	//Device Information Parameter
	_strDeviceCode		: STRING(51);		// Hardware Version Name from Device read acyclic	
	//Values read with acyclic FB
	_rTemperature		: REAL;				//24 P0-09 Heatsink Temperature ro RUN 40 ≙ 40 °C -10 - 150 –
	_rEnergy			: REAL;				//36 P0-26 kWh Meter ro RUN 100 ≙ 10.0 kWh 0 - N/A		(not possible with DE1)
    _rFreqMax  			: REAL; 			//129 P-01 f-max rw STOP 3000 ≙ 50.0 Hz P-02 - 300 Hz U16
    _rFreqMin 			: REAL; 			//130 P-02 f-min rw STOP 3000 ≙ 50.0 Hz 0 - P-01 U16
    _rTimeAcc 			: REAL; 			//131 P-03 t-acc rw RUN 300 ≙ 3.00 s 0.1 - 300 s U16
    _rTimeDec 			: REAL; 			//132 P-04 t-dec rw RUN 300 ≙ 3.00 s 0.1 - 300 s U16
    _rMotorNomVolt 		: REAL; 			//135 P-07 Motor Nom Voltage rw STOP 230 ≙ 230 V 50 - 500 V U16
    _rMotorNomCurr 		: REAL; 			//136 P-08 Motor Nom Current rw STOP 100 ≙ 10.0 A (10 - 100 %) x Ie U16
    _rMotorNomFreq 		: REAL; 			//137 P-09 Motor Nom Frequency rw STOP 50 ≙ 50 Hz 20 - 300 Hz U16
    _rMotorNomSpeed 	: REAL; 			//138 P-10 Motor Nom Speed rw STOP 1 ≙ 1 0 200 - 15000 rpm U16	

	//Single Device Infomation (https://www.eaton.com/content/dam/eaton/products/industrialcontrols-drives-automation-sensors/variable-frequency-drives/powerxl-dc1-variable-frequency-drives/communication-manual-for-variable-frequency-drives-variable-speed-starters-da1-dc1-de0-mn040018en.pdf)
	_eDriveType 				: teDriveTyp;	//the type of the connected Drive	
	_byFrameSize 				: BYTE;			//Frame size from connected Drive Frame size (FS) 1 = FS1, 2 = FS2, 3 = FS3, 4 = FS4
	_byVoltageClass 			: BYTE;			//Voltage class		0 = 115 V, 1 = 230 V, 2 = 230 V, 3 = 400 V
	_uiVoltage					: UINT;			//Voltage Unit V
	_rCurrentIr					: REAL;			//Current default value	in A
	_byNbInOutPhases 			: BYTE; 		//Input/output phases 1 or 3 phases on Iput and output side see table in documentation 
	_byPower 					: BYTE;			//Power from connected Drive
	_strTypeCode 				: STRING(9);	//create Typecode with read single Device Infomation
	_strNameDevice				: STRING;		//Name of the CanOpen Device from standard Object 1008h
	_SdoReadData 				: CIA405.SDO_READ_DATA ; 	//FB for Read SDO
	// Steps for reading asyclic Parameter
	_uiStep: UINT;
	_strSerialNbr: STRING;
END_VAR

SUPER^();

ACTION ACT_MapIO:
//Map SWD Pke value from Hardware structure to local Variable
IF _pstInput <> 0 THEN		
	//Loal Status Information from Drive
	stStatus.Readiness			:=_pstInput^.stStatusDrive.Readiness;
	stStatus.Operation			:=_pstInput^.stStatusDrive.Operation;
	stStatus.Rotation			:=_pstInput^.stStatusDrive.Rotation;
	stStatus.Fault				:=_pstInput^.stStatusDrive.Fault;
	stStatus.SetpointReached	:=_pstInput^.stStatusDrive.SetpointReached;				
	stStatus.ZeroSpeed			:=_pstInput^.stStatusDrive.ZeroSpeed;
	stStatus.SpeedControl		:=_pstInput^.stStatusDrive.SpeedControl;
	stStatus.HardwareEnable	:=_pstInput^.stStatusDrive.HardwareEnable;
	stStatus.ErrorCode			:=_pstInput^.stStatusDrive.ErrorCode;
	rActSpeed			:=INT_TO_REAL(_pstInput^.iMotorSpeed) / 10.0;
	rCurrent_A			:=INT_TO_REAL(_pstInput^.iCurrent) /10.0;
END_IF	
IF _pstOutput <> 0 THEN		
	//Commands for Drive
	 _pstOutput^.stCommandDrive.Operation			:=	stCommand.Operation	;	
	 _pstOutput^.stCommandDrive.Direction    		:=  stCommand.Direction		;	
	 _pstOutput^.stCommandDrive.ResetFault   		:=  stCommand.ResetFault		;	
	 _pstOutput^.stCommandDrive.FreeRunDown  		:=  stCommand.FreeRunDown	;	
	 _pstOutput^.stCommandDrive.QuickStop    		:=  stCommand.QuickStop		;	
	 _pstOutput^.stCommandDrive.FixedFrequencq		:=  stCommand.FixedFrequencq	;	
	 _pstOutput^.stCommandDrive.SetpointToZero		:=  stCommand.SetpointToZero	;
	 _pstOutput^.iSpeedReference						:= REAL_TO_INT(rSetpointSpeed *10);	
END_IF
END_ACTION

//Mapped real Hardware IO from GVL_IO to definied internal Structure and Interface
{attribute 'naming' := 'omit'} 
METHOD CyclicAction
VAR_INPUT
	{attribute 'analysis' := '-33'} 
	itfTimingController	: CBML.ITimingController; //Timing Controller for Check Time Out
END_VAR
VAR_OUTPUT
	//if xComplete or iErrorID <> 0 then the CleanupAction is reached
	xComplete	: BOOL;								//Normally never use
	iErrorID	: INT;								//Error is happen, Error Code 
END_VAR
//Call Cyclic Action form Device Base for standard error handling
SUPER^.CyclicAction(itfTimingController := itfTimingController ,xComplete=>xComplete, iErrorID =>iErrorID);

//Special Handling for different Fieldbus System
CASE _eBusType OF
	DED.BUS_TYPE.MODBUS_RTU:
		ACT_MapIO();
	ELSE
		ACT_MapIO();		
END_CASE

//Device specfic error code
IF stStatus.ErrorCode <> teDriveError.no_Flt THEN
	{analysis -34, -58, -130} //map device specific error code to a eaton uniqe global error code: offset for drive is 100
	eErrorCode := stStatus.ErrorCode + 100;
	{analysis +34, +58, +130}
END_IF

iErrorID := eErrorCode;
END_METHOD

//SET Rotation:  False = Clockwise rotating field (FWD),		TRUE = Anticlockwise rotating field (REV)
//GET Direction: False = Clockwise rotating field (FWD); 		TRUE = Anticlockwise rotating field (REV)
PROPERTY Direction : BOOL
GET
Direction := stStatus.Rotation;
END_GET
SET
stCommand.Direction := Direction;
END_SET
END_PROPERTY

//Error happen on Device
PROPERTY ErrorCode : teErrorCodeEaton
GET
// Implemntation of get 
{attribute 'analysis' := '-162'}
ErrorCode := eErrorCode;
END_GET
END_PROPERTY

//clean all values so that a restart is working fine again
METHOD ExitAction
VAR_INPUT
    xAfterCleanup : BOOL;
    xInCopyCode : BOOL;
END_VAR
SUPER^.ExitAction(xAfterCleanup:=xAfterCleanup, xInCopyCode :=xInCopyCode);

	IF _pstOutput <> 0 THEN
		 _pstOutput^.stCommandDrive.Operation			:=	FALSE	;	
		 _pstOutput^.stCommandDrive.Direction    		:=  FALSE	;	
		 _pstOutput^.stCommandDrive.ResetFault   		:=  FALSE	;	
		 _pstOutput^.stCommandDrive.FreeRunDown  		:=  FALSE	;	
		 _pstOutput^.stCommandDrive.QuickStop    		:=  TRUE	;	
		 _pstOutput^.stCommandDrive.FixedFrequencq		:=  FALSE	;	
		 _pstOutput^.stCommandDrive.SetpointToZero		:=  FALSE	;
		 _pstOutput^.iSpeedReference					:=  0;	
	END_IF
	_pstOutput 		:=0;		//Output Structure from DE1 Control Word
	_pstInput		:=0;		//Input  Structure from DE1 Status Word
	//Loal Status Information from Drive
	stStatus.Readiness			:=FALSE;				//False = Drive not ready; 						TRUE = ready FOR operation (READY)
	stStatus.Operation			:=FALSE;             //False = stop; 								TRUE = Operation (RUN)
	stStatus.Rotation			:=FALSE;             //False = Clockwise rotating field (FWD),		TRUE = Anticlockwise rotating field (REV)
	stStatus.Fault				:=FALSE;             //False = no error,								TRUE = Fault detected (FAULT)
	stStatus.SetpointReached	:=FALSE;             //False = Acceleration ramp 					TRUE = Frequency actual value equals setpoint input       							
	stStatus.ZeroSpeed			:=FALSE;             //False = -,									TRUE = Zero speed
	stStatus.SpeedControl		:=FALSE;             //False = Speed control deactivated,			TRUE = Speed control activated
	stStatus.HardwareEnable	:=FALSE;             //False = No coomunication,						TRUE = communication and Hardware okay
	stStatus.ErrorCode			:= teDriveError.no_Flt;		//Detailed Error Information Code
	rActSpeed			:= 0;				//Speed in Hz
	rCurrent_A			:= 0;				//Current in A
	//Values read with acyclic FB
	_rTemperature		:=0;				//24 P0-09 Heatsink Temperature ro RUN 40 ≙ 40 °C -10 - 150 –
	_rEnergy			:=0;				//36 P0-26 kWh Meter ro RUN 100 ≙ 10.0 kWh 0 - N/A		(not possible with DE1)
    _rFreqMax  			:=0; 				//129 P-01 f-max rw STOP 3000 ≙ 50.0 Hz P-02 - 300 Hz U16
    _rFreqMin 			:=0; 				//130 P-02 f-min rw STOP 3000 ≙ 50.0 Hz 0 - P-01 U16
    _rTimeAcc 			:=0; 				//131 P-03 t-acc rw RUN 300 ≙ 3.00 s 0.1 - 300 s U16
    _rTimeDec 			:=0; 				//132 P-04 t-dec rw RUN 300 ≙ 3.00 s 0.1 - 300 s U16
    _rMotorNomVolt 		:=0; 				//135 P-07 Motor Nom Voltage rw STOP 230 ≙ 230 V 50 - 500 V U16
    _rMotorNomCurr 		:=0; 				//136 P-08 Motor Nom Current rw STOP 100 ≙ 10.0 A (10 - 100 %) x Ie U16
    _rMotorNomFreq 		:=0; 				//137 P-09 Motor Nom Frequency rw STOP 50 ≙ 50 Hz 20 - 300 Hz U16
    _rMotorNomSpeed 	:=0; 				//138 P-10 Motor Nom Speed rw STOP 1 ≙ 1 0 200 - 15000 rpm U16
	
	//Commands for Drive
	stCommand.Operation		:=FALSE; 			//False = stop; 								TRUE = Operation
	stCommand.Direction		:=FALSE; 			//False = Clockwise rotating field (FWD); 		TRUE = Anticlockwise rotating field (REV)
	stCommand.ResetFault		:=FALSE; 			//False = No action,							TRUE = Fault Reset
	stCommand.FreeRunDown		:=FALSE; 			//False = No action,							TRUE = free run-down      							
	stCommand.QuickStop		:=FALSE; 			//False = No action,							TRUE = Quick stop (ramp)
	stCommand.FixedFrequencq	:=FALSE; 			//False = No action,							TRUE = Fixed frequency 1 (FF1)
	stCommand.SetpointToZero	:=FALSE; 			//False = No action,							TRUE = Overwrite setpoint value with 0
	rSetpointSpeed				:=0;				//Setpoint for Frequenzq Speed in Hz
	
	//Device Information Parameter
	_strDeviceCode				:='';				// Hardware Version Name from Device read acyclic

	//Single Device Infomation (https://www.eaton.com/content/dam/eaton/products/industrialcontrols-drives-automation-sensors/variable-frequency-drives/powerxl-dc1-variable-frequency-drives/communication-manual-for-variable-frequency-drives-variable-speed-starters-da1-dc1-de0-mn040018en.pdf)
	_eDriveType 				:= teDriveTyp.DE1;	//the type of the connected Drive	
	_byFrameSize 				:=0;			//Frame size from connected Drive Frame size (FS) 1 = FS1, 2 = FS2, 3 = FS3, 4 = FS4
	_byVoltageClass 			:=0;			//Voltage class		0 = 115 V, 1 = 230 V, 2 = 230 V, 3 = 400 V
	_uiVoltage					:=0;			//Voltage Unit V
	_rCurrentIr					:=0;			//Current default value	in A
	_byNbInOutPhases 			:=0; 		//Input/output phases 1 or 3 phases on Iput and output side see table in documentation 
	_byPower 					:=0;			//Power from connected Drive
	_strTypeCode 				:= '';	//create Typecode with read single Device Infomation
	
	
	// Steps for reading asyclic Parameter
	_uiStep:= 0;
	_strSerialNbr:='';
END_METHOD

//Property for get informatin about Fault and possible ack the Fault
PROPERTY Fault : BOOL
GET
Fault := stStatus.Fault;
END_GET
SET
stCommand.ResetFault := Fault;
END_SET
END_PROPERTY

//Property to set drive to a Fixed Frequeny
PROPERTY FixedFrequency : BOOL
SET
stCommand.FixedFrequencq := FixedFrequency;
END_SET
END_PROPERTY

//False = No action,							TRUE = free run-down 
PROPERTY FreeRunDown : BOOL
SET
stCommand.FreeRunDown := FreeRunDown;
END_SET
END_PROPERTY

//Method to get a Parameter from Drive
METHOD GetParameter : REAL
VAR_INPUT
	eParameter : teDriveParameter;	//Select the Parameter which you will get as return Value
END_VAR
CASE eParameter OF
	teDriveParameter.HeatsinkTemp : 	GetParameter := _rTemperature;
	teDriveParameter.MotorNomCurrent : 	GetParameter := _rMotorNomCurr;
	teDriveParameter.MotorNomFreq : 	GetParameter := _rMotorNomFreq;
	teDriveParameter.MotorNomSpeed :	GetParameter := _rMotorNomSpeed;
	teDriveParameter.MotorNomVoltage : 	GetParameter := _rMotorNomVolt;
	teDriveParameter.fmax : 			GetParameter := _rFreqMax;
	teDriveParameter.fmin : 			GetParameter := _rFreqMin;
	teDriveParameter.tacc :				GetParameter := _rTimeAcc;
	teDriveParameter.tdec : 			GetParameter := _rTimeDec;
ELSE
	GetParameter := 0.0;
END_CASE
END_METHOD

//GET: False = No coomunication,						TRUE = communication and Hardware okay
PROPERTY HardwareEnable : BOOL
GET
HardwareEnable := stStatus.HardwareEnable;
END_GET
END_PROPERTY

//Identification Modul Name
{attribute 'analysis' := '-23'} 
PROPERTY ModulName : STRING[51]
GET
// Implemntation of get 
{attribute 'analysis' := '-23-, 162'}
ModulName := _strTypeCode;
END_GET
END_PROPERTY

//SET: False = Drive not ready; 					TRUE = ready FOR operation (READY)
//GET: False = stop; 								TRUE = Operation
PROPERTY Operation : BOOL
GET
Operation := stStatus.Operation;
END_GET
SET
stCommand.Operation := Operation;
END_SET
END_PROPERTY

//Quick Stop in Control Structure
PROPERTY QuickStop : BOOL
SET
stCommand.QuickStop := QuickStop ;
END_SET
END_PROPERTY

//Property for get and set the ramp for start the drive
PROPERTY rAcceleration : Real
GET
rAcceleration := _rTimeAcc;
END_GET
SET
END_SET
END_PROPERTY

//actual current Value from Drive
PROPERTY rCurrent : REAL
GET
rCurrent := rCurrent_A;
END_GET
END_PROPERTY

//Property for get and set the deceleration ramp for stop the drive
PROPERTY rDeceleration : REAL
GET
rDeceleration := _rTimeDec;
END_GET
SET
END_SET
END_PROPERTY

//Get the Energy from Drive
PROPERTY rEnergy : REAL
GET
rEnergy := _rEnergy;
END_GET
END_PROPERTY

//Get and Set the Velocitiy from Drive
PROPERTY rVelocity : REAL
GET
rVelocity := rActSpeed;
END_GET
SET
rSetpointSpeed := rVelocity;
END_SET
END_PROPERTY

//False = Acceleration ramp 					TRUE = Frequency actual value equals setpoint input
PROPERTY SetpointReached : BOOL
GET
SetpointReached := stStatus.SetpointReached;
END_GET
END_PROPERTY

//Property for get speed control
//False = Speed control deactivated,			TRUE = Speed control activated
PROPERTY SpeedControl : BOOL
GET
SpeedControl := stStatus.SpeedControl;
END_GET
END_PROPERTY

//Initalization Routine
(*Init for Drive FB*)
{attribute 'naming' := 'omit'} 
METHOD StartAction
VAR_OUTPUT
	xComplete	: BOOL;		//Setting and Init Done, if the Variable is True the Method Cyclic will be called
	iErrorID	: INT;		//if Error is happen set ErrorID to Error Code, after that CLeanUp will Call with Error ID as an Input
END_VAR
VAR
	_pConfigParam : POINTER TO IoConfigParameter;
	_udiResult : UDINT;
	udiDataLength: UDINT;
END_VAR

//1000 00 Device Type Variable frequency drive – CANopen device ro 0 UNSIGNED32 
//1002 00 Manufacturer Status Register Emergency object fault log ro 00 UNSIGNED16  
//1008 00 Manufacturer Device Name The variable frequency drive's device name: DA1 ro DA1 STRING
//1009 00 Manufacturer Hardware Version Hardware version of the module ro 1.11 (Example) STRING
//100A 00 Manufacturer Software Version Software version of the module ro 1.00 (Example)STRING
//1018 	00 Identity Object General device information ro 04 UNSIGNED8 
//		01 Vendor ID Manufacturer: Eaton Industries GmbH ro 000001C7 UNSIGNED32 
//		02 Product Code Product Number ro 0 UNSIGNED32 
//		03 Revision Number Version ro 1.01 (Example) UNSIGNED32 
//		04 Serial Number Serial Number ro 00000001 (Example) UNSIGNED32
//Call Start Action form Device Base for standard caa device infomation
SUPER^.StartAction(xComplete=>xComplete, iErrorID =>iErrorID);
xComplete := FALSE;
//Check if In and Output is set
//Read the Parameter for the IO input pointer which is generate in the special devicedescription
_pConfigParam := IoStandard.ConfigGetParameter(pIoConnector:= _itfDevice.Connector, dwParameterId := 2147483649);
IF _pConfigParam <> 0 THEN
	_pbyInputAdress := IoStandard.ConfigGetParameterValuePointer(_pConfigParam, pResult:=ADR(_udiResult));
END_IF
IF _pbyInputAdress <> 0 THEN
	{analysis -19} //convert from input and output pointer to expected IO structure (control and status) 
	IF _eBusType = DED.BUS_TYPE.VEN_SPEC THEN
		_pstInput := _pbyInputAdress;
	ELSIF _eBusType = DED.BUS_TYPE.MODBUS_RTU THEN
		_pstInput := _pbyInputAdress;
	ELSE
		_pstInput := _pbyInputAdress;	
	END_IF	
ELSE
	eErrorCode := teErrorCodeEaton.InpAddressMiss; //wrong configuration
	iErrorID := TO_INT(eErrorCode);
END_IF
//Read the Parameter for the IO output pointer which is generate in the special devicedescription
_pConfigParam := IoStandard.ConfigGetParameter(pIoConnector:= _itfDevice.Connector, dwParameterId := 2147483648);
IF _pConfigParam <> 0 THEN
	_pbyOutputAdress := IoStandard.ConfigGetParameterValuePointer(_pConfigParam, pResult:=ADR(_udiResult));
END_IF
IF _pbyOutputAdress <> 0 THEN
	IF _eBusType = DED.BUS_TYPE.VEN_SPEC THEN
		_pstOutput := _pbyOutputAdress;
	ELSIF _eBusType = DED.BUS_TYPE.MODBUS_RTU THEN
		_pstOutput := _pbyOutputAdress;
	ELSE
		_pstOutput := _pbyOutputAdress;	
	END_IF		
	{analysis +19}		
ELSE
	eErrorCode := teErrorCodeEaton.OutAddressMiss; //wrong configuration 
	iErrorID := TO_INT(eErrorCode);
END_IF	



//Special Handling for different Fieldbus System
CASE _eBusType OF
	DED.BUS_TYPE.MODBUS_RTU: xComplete := TRUE;
	DED.BUS_TYPE.CANOPEN:  
		udiDataLength := SIZEOF (_strNameDevice);	
		_SdoReadData(
			NETWORK:= 1 , 
			ENABLE:= TRUE,  
			CONFIRM=> , 
			ERROR=> , 
			DEVICE:= DWORD_TO_USINT (_stDeviceInfo.idSystem),  
			INDEX:= 16#1008, 
			SUBINDEX:= , 
			MODE:= , 
			DATA:= ADR(_strNameDevice), 
			DATALENGTH:= udiDataLength, 
			ERRORINFO=> );
		IF 	_SdoReadData.CONFIRM THEN
			_strNameDevice := OSCAT_BASIC.MIRROR(str:= _strNameDevice);
			_SdoReadData(ENABLE := FALSE, DATALENGTH := udiDataLength);		
			IF Standard.FIND(STR1 := _strNameDevice, STR2 := 'DC1') > 0 THEN
				_eDriveType := teDriveTyp.DC1;
			ELSIF Standard.FIND(STR1 := _strNameDevice, STR2 := 'DA1') > 0  THEN
				_eDriveType := teDriveTyp.DA1;
			END_IF
			xComplete := TRUE;
		END_IF
		
END_CASE
END_METHOD

//Definition of Eaton Drive Type
PROPERTY TypeCode : teDriveTyp
GET
TypeCode := _eDriveType;
END_GET
END_PROPERTY

//Property for get and set the drive to Zero Speed
PROPERTY ZeroSpeed : BOOL
GET
ZeroSpeed := stStatus.ZeroSpeed;
END_GET
SET
stCommand.SetpointToZero := ZeroSpeed;
END_SET
END_PROPERTY

END_FUNCTION_BLOCK

// Interface/ITF_Drive
//Standard Interface for all Eaton Drives
INTERFACE ITF_Drive EXTENDS ITF_Base_MotorStarter

//Information which kind of Fieldbus is in use
PROPERTY eFieldbus : teFieldbus
GET
END_GET
END_PROPERTY

//Property for get informatin about Fault and possible ack the Fault
PROPERTY Fault : BOOL
GET
END_GET
SET
END_SET
END_PROPERTY

//Property to set drive to a Fixed Frequeny
PROPERTY FixedFrequency : BOOL
SET
END_SET
END_PROPERTY

//Free Run Down in Control Structure
PROPERTY FreeRunDown : BOOL
SET
END_SET
END_PROPERTY

//Method to get a Parameter from Drive
METHOD GetParameter : REAL
VAR_INPUT
	eParameter : teDriveParameter;
END_VAR
END_METHOD

//Property for get information if Drive is Enable
PROPERTY HardwareEnable : BOOL
GET
END_GET
END_PROPERTY

//Identification Modul Name
{attribute 'analysis' := '-23'} 
PROPERTY ModulName : STRING[51]
GET
END_GET
END_PROPERTY

//Quick Stop in Control Structure
PROPERTY QuickStop : BOOL
SET
END_SET
END_PROPERTY

//Property for get and set the ramp for start the drive
PROPERTY rAcceleration : Real
GET
END_GET
SET
END_SET
END_PROPERTY

//Property for get the actual current of the drive
PROPERTY rCurrent : REAL
GET
END_GET
END_PROPERTY

//Property for get and set the deceleration ramp for stop the drive
PROPERTY rDeceleration : REAL
GET
END_GET
SET
END_SET
END_PROPERTY

//Get the Energy from Drive
PROPERTY rEnergy : REAL
GET
END_GET
END_PROPERTY

//Get and Set the Velocitiy from Drive
PROPERTY rVelocity : REAL
GET
END_GET
SET
END_SET
END_PROPERTY

//Property for get information if drive the setpoint reached
PROPERTY SetpointReached : BOOL
GET
END_GET
END_PROPERTY

//Property for get speed control
PROPERTY SpeedControl : BOOL
GET
END_GET
END_PROPERTY

//Definition of Eaton Drive Type
PROPERTY TypeCode : teDriveTyp
GET
END_GET
END_PROPERTY

//Property for get and set the drive to Zero Speed
PROPERTY ZeroSpeed : BOOL
GET
END_GET
SET
END_SET
END_PROPERTY

END_INTERFACE

// Interface/ITF_Base_MotorStarter
//Interface for a Base Motor Starter
INTERFACE ITF_Base_MotorStarter EXTENDS __SYSTEM.IQueryInterface

//Property for get and set the direction of a Motor
PROPERTY Direction : BOOL
GET
END_GET
SET
END_SET
END_PROPERTY

//Error happen on Device
PROPERTY ErrorCode : teErrorCodeEaton
GET
END_GET
END_PROPERTY

//Set a Motor in operation or get Information if motor is running
PROPERTY Operation : BOOL
GET
END_GET
SET
END_SET
END_PROPERTY

END_INTERFACE

// FunctionBlock/FB_ErrorHandler
{attribute 'reflection'}
FUNCTION_BLOCK FB_ErrorHandler IMPLEMENTS I_ErroHandlerSubject
VAR_INPUT
END_VAR
VAR_OUTPUT
    astrActive : ARRAY [0..10] OF STRING[255];	//State from all existing FB
	uiNumOfActError : UINT;				
END_VAR
VAR
    {attribute 'instance-path'} 
    {attribute 'noinit'}
    _strName: STRING(255); 					// Instance path of the FB for Diagnostic
			
	_stInfoState : ARRAY [0..GVL_Const.MAX_Observer] OF tsCBMLInfo;	//State from all existing FB
	_stErrorState : ARRAY [0..GVL_Const.MAX_Observer] OF BOOL;			//State from all existing FB
	_uiNumberOfDevices : UINT;						//Number of Attached Devices
	uiHelp : UINT; 									//Help Variable for Loop
	
	//Help Variables for Attaching and read Information from Devices
	uiLoop : UINT;

END_VAR

//monitor all register Device by the IBehaviour Modell
_uiNumberOfDevices := 0;
FOR uiLoop := 0 TO GVL_Const.MAX_Observer DO  
	IF aritfObserver[uiLoop] <> 0 THEN
		_uiNumberOfDevices := _uiNumberOfDevices + 1;
		aritfObserver[uiLoop].GetModelState(	xCommit:= _stInfoState[uiLoop].xCommit, 
									xDone=> _stInfoState[uiLoop].xDone, 
									xBusy=> _stInfoState[uiLoop].xBusy, 
									xError=> _stInfoState[uiLoop].xError, 
									xAborted=> _stInfoState[uiLoop].xAborted, 
									iErrorID=> _stInfoState[uiLoop].iErrorID, 
									eState=> _stInfoState[uiLoop].eState);
		_stInfoState[uiLoop].strName := aritfObserver[uiLoop].GetName;							
		IF NOT _stErrorState[uiLoop] AND _stInfoState[uiLoop].xError THEN
			_stErrorState[uiLoop] := _stInfoState[uiLoop].xError;
			//Build Error String
			FOR uiHelp := 10 TO 1 BY -1 DO 
				IF uiHelp > 1 THEN
					astrActive[uiHelp] := astrActive [uiHelp-1];
				ELSIF uiHelp = 1 THEN
					uiNumOfActError := uiNumOfActError + 1;
 					astrActive[uiHelp] := CONCAT(CONCAT(CONCAT ('In FB ',_stInfoState[uiLoop].strName ),'the following error is activ:'), to_String (_stInfoState[uiLoop].iErrorID)) ;
				END_IF
			END_FOR
		ELSIF  _stErrorState[uiLoop] AND NOT _stInfoState[uiLoop].xError THEN
			_stErrorState[uiLoop] := _stInfoState[uiLoop].xError;
			//Build Error String
			FOR uiHelp := 10 TO 1 BY -1 DO 
				IF uiHelp > 1 THEN
					astrActive[uiHelp] := astrActive [uiHelp-1];
				ELSIF uiHelp = 1 THEN
					uiNumOfActError := uiNumOfActError - 1;
 					astrActive[uiHelp] := CONCAT(CONCAT(CONCAT ('In FB ',_stInfoState[uiLoop].strName ),'the following error is deactiv:'),to_String (_stInfoState[uiLoop].iErrorID)) ;
				END_IF
			END_FOR
		END_IF					
    END_IF
END_FOR

METHOD AttachDevice 
(*Register a Device by the BehaiourModel Interface*)
VAR_INPUT
	(*Device which will be monitor from Error Handler*)
	IDevice	: IBasicBehaviour;
END_VAR

VAR
	uiLoop: UINT;
END_VAR
FOR uiLoop := 1 TO GVL_Const.MAX_Observer DO
	IF IDevice <> 0 AND aritfObserver[uiLoop]= 0 THEN
		aritfObserver[uiLoop] := IDevice;
		EXIT;
	END_IF
END_FOR
END_METHOD

METHOD DetachDevice 
(*Unregister a Device by the BehaiourModel Interface*)
VAR_INPUT
	(*Device which will be deleted from the monitor Error Handler list*)
	IDevice	: IBasicBehaviour;
END_VAR

VAR
	uiLoop: UINT;
END_VAR
FOR uiLoop := 0 TO GVL_Const.MAX_Observer DO
	IF IDevice <> 0 AND .aritfObserver[uiLoop]= IDevice THEN
		aritfObserver[uiLoop] := 0;
		EXIT;
	END_IF
END_FOR
END_METHOD

END_FUNCTION_BLOCK

// Interface/I_ErroHandlerSubject
INTERFACE I_ErroHandlerSubject EXTENDS __System.IQueryInterface

METHOD AttachDevice 
(*Register a Device by the BehaiourModel Interface*)
VAR_INPUT
	(*Device which will be monitor from Error Handler*)
	IDevice	: IBasicBehaviour;
END_VAR
END_METHOD

METHOD DetachDevice 
(*Unregister a Device by the BehaiourModel Interface*)
VAR_INPUT
	(*Device which will be deleted from the monitor Error Handler list*)
	IDevice	: IBasicBehaviour;
END_VAR
END_METHOD

END_INTERFACE

// Device/Application/InputData
FUNCTION_BLOCK InputData
VAR_INPUT
	itfDevice : DED.IDevice;
	dwParam : DWORD;
END_VAR
VAR_OUTPUT
	dwData : DWORD;
END_VAR
VAR
	pConfigParam : POINTER TO IoConfigParameter;
	udiResult : UDINT;
	Connector: POINTER TO DED.IoConfigConnector;
END_VAR

Connector := itfDevice.Connector;

pConfigParam := IoStandard.ConfigGetParameter(itfDevice.Connector, dwParam);
IF pConfigParam <> 0 THEN
	dwData := IoStandard.ConfigGetParameterValueDword(pConfigParam, pResult:=ADR(udiResult));
END_IF

END_FUNCTION_BLOCK

// Device/Application/PRG_PLC
PROGRAM PRG_PLC
VAR
		MyMotor : FB_Drive;
END_VAR

MyMotor(xEnable := TRUE, itfHW_Node := DC1); // FB_Drive

END_PROGRAM
